// TIA Portal project "LAb1.1" (V16)

(* hardware
DEVICE "S7-1200 station_1"  S7-1200 Station
   slot 0: "Rack_0"  S7-1200 Rack  Rack  V1.0
   slot 1: "PLC_1"  CPU 1211C AC/DC/Rly  6ES7 211-1BE40-0XB0  V4.4
DEVICE "HMI_1"  KTP700 Basic PN
   slot 0: "HMI_1"  KTP700 Basic PN  6AV2 123-2GB03-0AX0  16.0.0.0
   slot 1: "HMI_RT_1"  KTP700 Basic PN  6AV2 123-2GB03-0AX0  16.0.0.0
   slot 5: "HMI_1.IE_CP_1"  PROFINET Interface  16.0.0.0
      slot 1: "PROFINET Interface_1"  PROFINET Interface
         slot 1: "Port_1"  Port
DEVICE "HMI_2"  KTP700 Basic PN
   slot 0: "HMI_2"  KTP700 Basic PN  6AV2 123-2GB03-0AX0  15.1.0.0
   slot 1: "HMI_RT_2"  KTP700 Basic PN  6AV2 123-2GB03-0AX0  15.1.0.0
   slot 5: "HMI_2.IE_CP_1"  PROFINET Interface  15.0.1.0
      slot 1: "PROFINET Interface_1"  PROFINET Interface
         slot 1: "Port_1"  Port
*)

// ===== PLC "PLC_1"  CPU 1211C AC/DC/Rly =====

VAR_GLOBAL   // PLC tag table "Default tag table"
   "START" AT %M0.2 : Bool;
   "LAMP" AT %Q0.1 : Bool;
   "LAMP_1" AT %M0.0 : Bool;
   "T1_INPUT" AT %MD2 : DInt;
   "T2_INPUT" AT %MD10 : DInt;
   "T1_INPUT_RESULT" AT %MD6 : DInt;
   "T2_INPUT_RESULT" AT %MD14 : DInt;
   "T1_HMI" AT %MD18 : DInt;
   "T2_HMI" AT %MD22 : DInt;
   "STOP" AT %M0.3 : Bool;
END_VAR

// folder: System blocks/Program resources

DATA_BLOCK "Timer1"   // DB3
{ S7_Optimized_Access := 'TRUE' }
AUTHOR : Simatic
FAMILY : IEC
NAME : IEC_TMR
VERSION : 1.0
// stored: InstanceOfName IEC_TIMER
"IEC_TIMER"
BEGIN
END_DATA_BLOCK

DATA_BLOCK "Timer2"   // DB4
{ S7_Optimized_Access := 'TRUE' }
AUTHOR : Simatic
FAMILY : IEC
NAME : IEC_TMR
VERSION : 1.0
// stored: InstanceOfName IEC_TIMER
"IEC_TIMER"
BEGIN
END_DATA_BLOCK

// folder: (top level)

ORGANIZATION_BLOCK "Main"   // OB1, LAD, ProgramCycle
TITLE = "Main Program Sweep (Cycle)"
{ S7_Optimized_Access := 'TRUE' }
VERSION : 0.1
   VAR_INPUT
      Initial_Call : Bool;   // Initial call of this OB
      Remanence : Bool;   // =True, if remanent data are available
   END_VAR
BEGIN

REGION Network 1
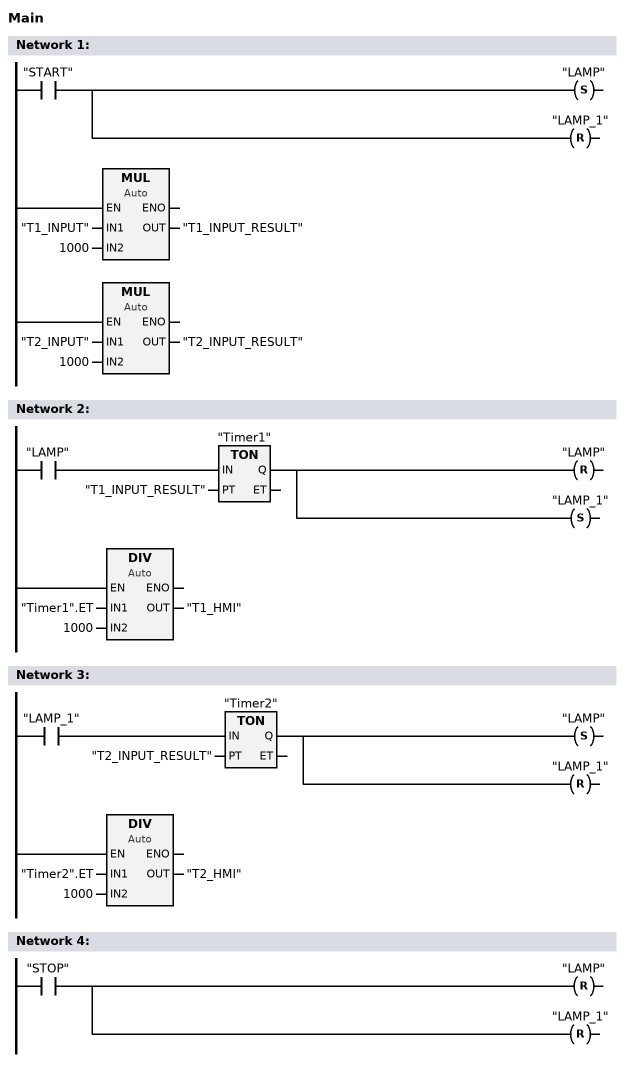
   RUNG wire#powerrail
      Contact( "START" )
      wire#w1
      S_Coil( "LAMP" )
   END_RUNG
   RUNG wire#w1
      R_Coil( "LAMP_1" )
   END_RUNG
   RUNG wire#powerrail
      Mul(in1 := "T1_INPUT", in2 := 1000, out => "T1_INPUT_RESULT")
   END_RUNG
   RUNG wire#powerrail
      Mul(in1 := "T2_INPUT", in2 := 1000, out => "T2_INPUT_RESULT")
   END_RUNG
   // the same network as SCL:
   IF "START" THEN
       "LAMP" := TRUE;
       "LAMP_1" := FALSE;
   END_IF;
   "T1_INPUT_RESULT" := "T1_INPUT" * 1000;
   "T2_INPUT_RESULT" := "T2_INPUT" * 1000;
END_REGION

REGION Network 2
   "Timer1".TON(IN := "LAMP", PT := "T1_INPUT_RESULT");
   IF "Timer1".Q THEN
       "LAMP" := FALSE;
       "LAMP_1" := TRUE;
   END_IF;
   "T1_HMI" := "Timer1".ET / 1000;
END_REGION

REGION Network 3
   "Timer2".TON(IN := "LAMP_1", PT := "T2_INPUT_RESULT");
   IF "Timer2".Q THEN
       "LAMP" := TRUE;
       "LAMP_1" := FALSE;
   END_IF;
   "T2_HMI" := "Timer2".ET / 1000;
END_REGION

REGION Network 4
   RUNG wire#powerrail
      Contact( "STOP" )
      wire#w1
      R_Coil( "LAMP" )
   END_RUNG
   RUNG wire#w1
      R_Coil( "LAMP_1" )
   END_RUNG
   // the same network as SCL:
   IF "STOP" THEN
       "LAMP" := FALSE;
       "LAMP_1" := FALSE;
   END_IF;
END_REGION
END_ORGANIZATION_BLOCK

(* ===== HMI "HMI_RT_1" =====
system functions are stored by id; their names below are inferred from use
connection "HMI_Connection_1": ETHERNET, SMART_S7_1200_OMS
connection "HMI_Connection_2": ETHERNET, SMART_S7_1200_OMS
connection "HMI_Connection_3": ETHERNET, SMART_S7_1200_OMS

HMI tags "Default tag table"
   "START" : Bool = PLC START AT %M0.2, 1 s
   "STOP" : Bool = PLC STOP AT %M0.3, 1 s
   "LAMP_1" : Bool = PLC LAMP_1 AT %M0.0, 1 s
   "LAMP" : Bool = PLC LAMP AT %Q0.1, 1 s
   "T1_INPUT" : DInt = PLC T1_INPUT AT %MD2, 1 s
   "T2_INPUT" : DInt = PLC T2_INPUT AT %MD10, 1 s
   "T2_INPUT_RESULT" : DInt = PLC T2_INPUT_RESULT AT %MD14, 1 s
   "T1_HMI" : DInt = PLC T1_HMI AT %MD18, 1 s
   "T2_HMI" : DInt = PLC T2_HMI AT %MD22, 1 s

screen "Root screen" 800x480, template "Template_1"
   Button "HmiScreenItemData_1" at 36,36 size 159x47; TextOff 'System screens'; PictureOff "Navigates to System screens for KTP700 Basic+ PN 16.0.0.0"; PictureOn "Navigates to System screens for KTP700 Basic+ PN 16.0.0.0"
      on Release: ActivateScreen("System screens", 0)
   Button "Button_1" at 146,146 size 96x32; TextOff 'Start'
      on Press: SetBit("START")
      on Release: ResetBit("START")
   Button "Button_2" at 147,188 size 96x32; TextOff 'Stop'
      on Press: SetBit("STOP")
      on Release: ResetBit("STOP")
   Circle "Circle_1" at 296,137 size 83x83
      Appearance <- "LAMP"
   TextField "Text field_1" at 117,259 size 147x23; Text 'TIMER SETTINGS'
   TextField "Text field_2" at 331,258 size 126x23; Text 'TIME ELAPSED'
   TextField "Text field_3" at 116,299 size 53x23; Text 'T1 (s)'
   TextField "Text field_4" at 117,333 size 53x23; Text 'T2 (s)'
   TextField "Text field_5" at 315,299 size 53x23; Text 'T1 (s)'
   TextField "Text field_6" at 316,333 size 53x23; Text 'T2 (s)'
   IOField "I/O field_1" at 181,293 size 96x32; FormatPattern s9999999999
      Appearance <- "T1_INPUT"
      ProcessValue <- "T1_INPUT"
   IOField "I/O field_2" at 181,330 size 96x32; FormatPattern s9999999999
      Appearance <- "T2_INPUT"
      ProcessValue <- "T2_INPUT"
   IOField "I/O field_3" at 370,290 size 96x32; FormatPattern s9999999999
      Appearance <- "T1_HMI"
      ProcessValue <- "T1_HMI"
   IOField "I/O field_4" at 370,327 size 96x32; FormatPattern s9999999999
      Appearance <- "T2_HMI"
      ProcessValue <- "T2_HMI"
   Circle "Circle_2" at 424,137 size 83x83
      Appearance <- "LAMP_1"

screen "System screens" 800x480, template "Template_1"
   Button "Back" at 1,1 size 159x47; TextOff 'Back'
      on Release: ActivateScreen("Root screen", 0)
   Button "HmiScreenItemData" at 36,95 size 159x47; TextOff 'SIMATIC PLC system diagnos...'; PictureOff "Navigates to SIMATIC PLC system diagnostics for KTP700 Basic+ PN 16.0.0.0"; PictureOn "Navigates to SIMATIC PLC system diagnostics for KTP700 Basic+ PN 16.0.0.0"
      on Release: ActivateScreen("SIMATIC PLC system diagnostics", 0)
   Button "HmiScreenItemData_1" at 36,154 size 159x47; TextOff 'Project information'; PictureOff "Navigates to Project information for KTP700 Basic+ PN 16.0.0.0"; PictureOn "Navigates to Project information for KTP700 Basic+ PN 16.0.0.0"
      on Release: ActivateScreen("Project information", 0)
   Button "HmiScreenItemData_2" at 36,213 size 159x47; TextOff 'User administration'; PictureOff "Navigates to User administration for KTP700 Basic+ PN 16.0.0.0"; PictureOn "Navigates to User administration for KTP700 Basic+ PN 16.0.0.0"
      on Release: ActivateScreen("User administration", 0)
   Button "HmiScreenItemData_3" at 36,272 size 159x47; TextOff 'System information'; PictureOff "Navigates to System information for KTP700 Basic+ PN 16.0.0.0"; PictureOn "Navigates to System information for KTP700 Basic+ PN 16.0.0.0"
      on Release: ActivateScreen("System information", 0)
   Button "HmiScreenItemData_4" at 36,331 size 159x47; TextOff 'Different jobs'; PictureOff "Navigates to Different jobs for KTP700 Basic+ PN 16.0.0.0"; PictureOn "Navigates to Different jobs for KTP700 Basic+ PN 16.0.0.0"
      on Release: ActivateScreen("Different jobs", 0)

screen "SIMATIC PLC system diagnostics" 800x480, template "Template_1"
   SysDiagControl "HmiScreenItemData" at 1,49 size 796x423
   Button "Back" at 1,1 size 159x47; TextOff 'Back'
      on Release: ActivateScreen("System screens", 0)

screen "Project information" 800x480, template "Template_1"
   TextField "HmiScreenItemData" at 35,51 size 171x28; Text 'Project name:'
   TextField "HmiScreenItemData_1" at 241,51 size 524x28; Text 'LAb1.1'
   TextField "HmiScreenItemData_2" at 35,81 size 171x28; Text 'Created on:'
   TextField "HmiScreenItemData_3" at 241,81 size 524x28; Text '6/8/2026 9:46:48 AM'
   TextField "HmiScreenItemData_4" at 35,111 size 171x28; Text 'Author:'
   TextField "HmiScreenItemData_5" at 241,111 size 524x28; Text 'Khoa'
   TextField "HmiScreenItemData_6" at 35,141 size 171x28; Text 'Description:'
   TextField "HmiScreenItemData_7" at 241,141 size 524x28; Text '(not configured)'
   Button "Back" at 1,1 size 159x47; TextOff 'Back'
      on Release: ActivateScreen("System screens", 0)

screen "User administration" 800x480, template "Template_1"
   UserView "HmiScreenItemData" at 1,49 size 796x423
   Button "Back" at 1,1 size 159x47; TextOff 'Back'
      on Release: ActivateScreen("System screens", 0)

screen "System information" 800x480, template "Template_1"
   TextField "HmiScreenItemData" at 35,51 size 171x28; Text 'HMI device type:'
   TextField "HmiScreenItemData_1" at 241,51 size 524x28; Text 'KTP700 Basic+ PN 16.0.0.0'
   TextField "HmiScreenItemData_2" at 35,81 size 171x28; Text 'Connection:'
   TextField "HmiScreenItemData_3" at 241,81 size 524x28; Text 'PROFINET (X1)'
   TextField "HmiScreenItemData_4" at 35,111 size 171x28; Text 'PLC:'
   TextField "HmiScreenItemData_5" at 241,111 size 524x28; Text 'SIMATIC S7 1200'
   Button "Back" at 1,1 size 159x47; TextOff 'Back'
      on Release: ActivateScreen("System screens", 0)

screen "Different jobs" 800x480, template "Template_1"
   Button "Online" at 36,95 size 159x47; TextOff 'Online'
      on Release: function_bb44b551(0)
   Button "Offline" at 36,154 size 159x47; TextOff 'Offline'
      on Release: function_bb44b551(1)
   Button "Transfer" at 36,213 size 159x47; TextOff 'Transfer'
      on Release: function_bb44b551(2)
   Button "Toggle language" at 36,272 size 159x47; TextOff 'Toggle language'
      on Release: function_fb9197e8(-1)
   Button "Stop Runtime" at 36,331 size 159x47; TextOff 'Stop Runtime'
      on Release: StopRuntime(0)
   Button "Back" at 1,1 size 159x47; TextOff 'Back'
      on Release: ActivateScreen("System screens", 0)
*)

(* ===== HMI "HMI_RT_2" =====
system functions are stored by id; their names below are inferred from use
connection "HMI_Connection_4": ETHERNET, SMART_S7_1200_OMS
connection "HMI_Connection_5": ETHERNET, SMART_S7_1200_OMS

HMI tags "Default tag table"
   "START" : Bool = PLC START AT %M0.2, 1 s
   "LAMP" : Bool = PLC LAMP AT %Q0.1, 1 s
   "LAMP_1" : Bool = PLC LAMP_1 AT %M0.0, 1 s
   "T1_INPUT" : DInt = PLC T1_INPUT AT %MD2, 1 s
   "T2_INPUT" : DInt = PLC T2_INPUT AT %MD10, 1 s
   "T1_INPUT_RESULT" : DInt = PLC T1_INPUT_RESULT AT %MD6, 1 s
   "T2_INPUT_RESULT" : DInt = PLC T2_INPUT_RESULT AT %MD14, 1 s
   "T1_HMI" : DInt = PLC T1_HMI AT %MD18, 1 s
   "T2_HMI" : DInt = PLC T2_HMI AT %MD22, 1 s
   "STOP" : Bool = PLC STOP AT %M0.3, 1 s

screen "Root screen" 800x480, template "Template_1"
   TextField "HmiScreenItemData" at 80,225 size 640x25; Text 'Welcome to HMI_2 (KTP700 Basic+ PN)!'
   Button "HmiScreenItemData_1" at 36,36 size 159x47; TextOff 'System screens'; PictureOff "Navigates to System screens for KTP700 Basic+ PN 15.1.0.0"; PictureOn "Navigates to System screens for KTP700 Basic+ PN 15.1.0.0"
      on Release: ActivateScreen("System screens", 0)
   Button "Button_1" at 146,146 size 96x32; TextOff 'Start'
      on Release: ResetBit("START")
      on Press: SetBit("START")
   Button "Button_2" at 147,188 size 96x32; TextOff 'Stop'
      on Release: ResetBit("STOP")
      on Press: SetBit("STOP")
   Circle "Circle_1" at 296,137 size 83x83
      Appearance <- "LAMP"
   TextField "Text field_1" at 117,259 size 147x23; Text 'TIMER SETTINGS'
   TextField "Text field_2" at 331,258 size 126x23; Text 'TIME ELAPSED'
   TextField "Text field_3" at 116,299 size 53x23; Text 'T1 (s)'
   TextField "Text field_4" at 117,333 size 53x23; Text 'T2 (s)'
   TextField "Text field_5" at 315,299 size 53x23; Text 'T1 (s)'
   TextField "Text field_6" at 316,333 size 53x23; Text 'T2 (s)'
   IOField "I/O field_1" at 181,293 size 96x32; FormatPattern s9999999999
      ProcessValue <- "T1_INPUT"
      Appearance <- "T1_INPUT"
   IOField "I/O field_2" at 181,330 size 96x32; FormatPattern s9999999999
      ProcessValue <- "T2_INPUT"
      Appearance <- "T2_INPUT"
   IOField "I/O field_3" at 370,290 size 96x32; FormatPattern s9999999999
      ProcessValue <- "T1_HMI"
      Appearance <- "T1_HMI"
   IOField "I/O field_4" at 370,327 size 96x32; FormatPattern s9999999999
      ProcessValue <- "T2_HMI"
      Appearance <- "T2_HMI"
   Circle "Circle_2" at 424,137 size 83x83
      Appearance <- "LAMP_1"

screen "System screens" 800x480, template "Template_1"
   Button "Back" at 1,1 size 159x47; TextOff 'Back'
      on Release: ActivateScreen("Root screen", 0)
   Button "HmiScreenItemData" at 36,95 size 159x47; TextOff 'SIMATIC PLC system diagnos...'; PictureOff "Navigates to SIMATIC PLC system diagnostics for KTP700 Basic+ PN 15.1.0.0"; PictureOn "Navigates to SIMATIC PLC system diagnostics for KTP700 Basic+ PN 15.1.0.0"
      on Release: ActivateScreen("SIMATIC PLC system diagnostics", 0)
   Button "HmiScreenItemData_1" at 36,154 size 159x47; TextOff 'Project information'; PictureOff "Navigates to Project information for KTP700 Basic+ PN 15.1.0.0"; PictureOn "Navigates to Project information for KTP700 Basic+ PN 15.1.0.0"
      on Release: ActivateScreen("Project information", 0)
   Button "HmiScreenItemData_2" at 36,213 size 159x47; TextOff 'User administration'; PictureOff "Navigates to User administration for KTP700 Basic+ PN 15.1.0.0"; PictureOn "Navigates to User administration for KTP700 Basic+ PN 15.1.0.0"
      on Release: ActivateScreen("User administration", 0)
   Button "HmiScreenItemData_3" at 36,272 size 159x47; TextOff 'System information'; PictureOff "Navigates to System information for KTP700 Basic+ PN 15.1.0.0"; PictureOn "Navigates to System information for KTP700 Basic+ PN 15.1.0.0"
      on Release: ActivateScreen("System information", 0)
   Button "HmiScreenItemData_4" at 36,331 size 159x47; TextOff 'Different jobs'; PictureOff "Navigates to Different jobs for KTP700 Basic+ PN 15.1.0.0"; PictureOn "Navigates to Different jobs for KTP700 Basic+ PN 15.1.0.0"
      on Release: ActivateScreen("Different jobs", 0)

screen "SIMATIC PLC system diagnostics" 800x480, template "Template_1"
   SysDiagControl "HmiScreenItemData" at 1,49 size 796x423
   Button "Back" at 1,1 size 159x47; TextOff 'Back'
      on Release: ActivateScreen("System screens", 0)

screen "Project information" 800x480, template "Template_1"
   TextField "HmiScreenItemData" at 35,51 size 171x28; Text 'Project name:'
   TextField "HmiScreenItemData_1" at 241,51 size 524x28; Text 'LAb1.1'
   TextField "HmiScreenItemData_2" at 35,81 size 171x28; Text 'Created on:'
   TextField "HmiScreenItemData_3" at 241,81 size 524x28; Text '6/8/2026 9:46:48 AM'
   TextField "HmiScreenItemData_4" at 35,111 size 171x28; Text 'Author:'
   TextField "HmiScreenItemData_5" at 241,111 size 524x28; Text 'Khoa'
   TextField "HmiScreenItemData_6" at 35,141 size 171x28; Text 'Description:'
   TextField "HmiScreenItemData_7" at 241,141 size 524x28; Text '(not configured)'
   Button "Back" at 1,1 size 159x47; TextOff 'Back'
      on Release: ActivateScreen("System screens", 0)

screen "User administration" 800x480, template "Template_1"
   UserView "HmiScreenItemData" at 1,49 size 796x423
   Button "Back" at 1,1 size 159x47; TextOff 'Back'
      on Release: ActivateScreen("System screens", 0)

screen "System information" 800x480, template "Template_1"
   TextField "HmiScreenItemData" at 35,51 size 171x28; Text 'HMI device type:'
   TextField "HmiScreenItemData_1" at 241,51 size 524x28; Text 'KTP700 Basic+ PN 15.1.0.0'
   TextField "HmiScreenItemData_2" at 35,81 size 171x28; Text 'Connection:'
   TextField "HmiScreenItemData_3" at 241,81 size 524x28; Text 'PROFINET (X1)'
   TextField "HmiScreenItemData_4" at 35,111 size 171x28; Text 'PLC:'
   TextField "HmiScreenItemData_5" at 241,111 size 524x28; Text 'SIMATIC S7 1200'
   Button "Back" at 1,1 size 159x47; TextOff 'Back'
      on Release: ActivateScreen("System screens", 0)

screen "Different jobs" 800x480, template "Template_1"
   Button "Online" at 36,95 size 159x47; TextOff 'Online'
      on Release: function_bb44b551(0)
   Button "Offline" at 36,154 size 159x47; TextOff 'Offline'
      on Release: function_bb44b551(1)
   Button "Transfer" at 36,213 size 159x47; TextOff 'Transfer'
      on Release: function_bb44b551(2)
   Button "Toggle language" at 36,272 size 159x47; TextOff 'Toggle language'
      on Release: function_fb9197e8(-1)
   Button "Stop Runtime" at 36,331 size 159x47; TextOff 'Stop Runtime'
      on Release: StopRuntime(0)
   Button "Back" at 1,1 size 159x47; TextOff 'Back'
      on Release: ActivateScreen("System screens", 0)
*)